(* CODESYS project FU_sConcat7BO.xml

Project tree, tasks and I/O mapping:
  function FU_sConcat7BO [ST]
*)

// FU_sConcat7BO
//This functions combines seven strings
//This is the big output version, it has no limits to input or output size
//The wOutSize must be correct otherwise the function can write to unwanted addresses
// |**Version**|**Author**| **Date** |**Changes**
// | 1         | NSN      | 29-11-19 | Creation
// | 2         | NSN      | 14-10-21 | Changed to pointer based
FUNCTION FU_sConcat7BO : BOOL
VAR_IN_OUT
	sOut		:POINTER TO EASCII;			//Output String
END_VAR
VAR_INPUT
	s1			:STRING(255);			//Input String1
	s2			:STRING(255);			//Input String2
	s3			:STRING(255);			//Input String3
	s4			:STRING(255);			//Input String4
	s5			:STRING(255);			//Input String5
	s6			:STRING(255);			//Input String6
	s7			:STRING(255);			//Input String7
	wOutSize	:WORD;				//Output String Size
END_VAR

FU_sConcat7BIBO(sOut:=sOut,s1:=ADR(s1),s2:=ADR(s2),s3:=ADR(s3),s4:=ADR(s4),s5:=ADR(s5),s6:=ADR(s6),s7:=ADR(s7),wOutSize:=wOutSize);

END_FUNCTION
